// TIA Portal project "Project4" (V15.1)

(* hardware
DEVICE "S7-1200 station_2"  S7-1200 Station
   slot 0: "Rack_0"  S7-1200 Rack  Rack  V1.0
   slot 1: "CLP2_TESTING"  CPU 1214C DC/DC/DC  6ES7 214-1AG40-0XB0  V4.2
      slot 3: "AQ 1x12BIT_1"  AQ1 signal board  6ES7 232-4HA30-0XB0  V1.0
   slot 2: "DI 8/DQ 8x24VDC_1"  SM 1223 DI8/DQ8 x 24VDC  6ES7 223-1BH30-0XB0  V1.0
*)

// ===== PLC "CLP2_TESTING"  CPU 1214C DC/DC/DC =====

VAR_GLOBAL   // PLC tag table "Default tag table"
   "PART_AV" AT %I0.0 : Bool;
   "B2" AT %I0.1 : Bool;
   "B4" AT %I0.2 : Bool;
   "B5" AT %I0.3 : Bool;
   "1B1" AT %I0.4 : Bool;
   "1B2" AT %I0.5 : Bool;
   "2B1" AT %I0.6 : Bool;
   "IP_FI" AT %I0.7 : Bool;
   "Bot_Start" AT %I8.0 : Bool;
   "Bot_Stop" AT %I8.1 : Bool;
   "Bot_Reset" AT %I8.3 : Bool;
   "Desce_Elevador" AT %Q0.0 : Bool;
   "Sobe_Elevador" AT %Q0.1 : Bool;
   "Empurra_Peça" AT %Q0.2 : Bool;
   "Rampa" AT %Q0.3 : Bool;
   "IP_N_FO" AT %Q0.7 : Bool;
   "LED_Start" AT %Q8.0 : Bool;
   "LED_Reset" AT %Q8.1 : Bool;
   "LED_Q1" AT %Q8.2 : Bool;
   "LED_Q2" AT %Q8.3 : Bool;
   "void" AT %M57.0 : Bool;
   "Chega_Peça" AT %M0.0 : Bool;
   "Subida_Liberada" AT %M0.1 : Bool;
   "void2" AT %M57.1 : Bool;
   "Elevador_Em_Cima" AT %M0.3 : Bool;
   "void3" AT %M57.2 : Bool;
   "Elevador_Embaixo" AT %M0.4 : Bool;
   "void4" AT %M57.3 : Bool;
   "Pistão_Recuou" AT %M0.5 : Bool;
   "void5" AT %M57.4 : Bool;
   "Altura_Certa" AT %M0.6 : Bool;
   "Prox.Bancada_Liberou" AT %M0.7 : Bool;
   "void6" AT %M57.5 : Bool;
   "void7" AT %M57.6 : Bool;
   "void8" AT %M57.7 : Bool;
   "Start" AT %M1.0 : Bool;
   "Reset" AT %M1.1 : Bool;
   "Stop" AT %M1.2 : Bool;
   "Elevador_Subindo" AT %M2.0 : Bool;
   "Testando_Altura" AT %M2.1 : Bool;
   "Elevador_Descendo_c_Peça" AT %M2.2 : Bool;
   "Empurrando_Peça" AT %M2.3 : Bool;
   "Elevador_Descendo_Vazio" AT %M2.4 : Bool;
   "Descartando_Peça" AT %M2.5 : Bool;
   "Elevador_Livre" AT %M2.6 : Bool;
   "Contador_Descarte" AT %MW4 : Int;
   "Rampa_Desl" AT %M3.0 : Bool;
   "Rampa_Lig" AT %M3.1 : Bool;
   "Prox_Bancada_Livre" AT %M3.2 : Bool;
   "Parado" AT %M3.3 : Bool;
   "Resetando_Elevador" AT %M3.4 : Bool;
   "Pronto" AT %M3.5 : Bool;
   "Tem_Peça" AT %M2.7 : Bool;
   "T1" AT %M4.0 : Bool;
   "T2" AT %M4.1 : Bool;
   "T3" AT %M4.2 : Bool;
   "T4" AT %M4.3 : Bool;
   "T5" AT %M4.4 : Bool;
   "T6" AT %M4.5 : Bool;
   "T7" AT %M4.6 : Bool;
   "T8" AT %M6.0 : Bool;
   "T9" AT %M6.1 : Bool;
   "T10" AT %M6.2 : Bool;
   "T11" AT %M6.3 : Bool;
   "T12" AT %M6.4 : Bool;
   "T13" AT %M6.5 : Bool;
   "T14" AT %M6.6 : Bool;
   "T15" AT %M6.7 : Bool;
   "T16" AT %M7.0 : Bool;
   "T17" AT %M7.1 : Bool;
   "T18" AT %M7.2 : Bool;
   "T19" AT %M7.3 : Bool;
   "T20" AT %M7.4 : Bool;
   "T21" AT %M7.5 : Bool;
   "T22" AT %M7.6 : Bool;
   "T23" AT %M7.7 : Bool;
   "T24" AT %M8.0 : Bool;
   "T0" AT %M8.1 : Bool;
   "Fim_Reset" AT %M8.2 : Bool;
   "T25" AT %M8.3 : Bool;
   "Memo_Inicialização" AT %M58.0 : Bool;
   "T26" AT %M8.4 : Bool;
   "Resetando_Pistão" AT %M3.6 : Bool;
   "T27" AT %M8.5 : Bool;
   "Tag_1" AT %M58.1 : Bool;
   "Pistão_Recuado" AT %M58.2 : Bool;
END_VAR

// folder: System blocks/Program resources

DATA_BLOCK "IEC_Timer_0_DB_2"   // DB1
{ S7_Optimized_Access := 'TRUE' }
AUTHOR : Simatic
FAMILY : IEC
NAME : IEC_TMR
VERSION : 1.0
// stored: InstanceOfName IEC_TIMER
"IEC_TIMER"
BEGIN
END_DATA_BLOCK

DATA_BLOCK "IEC_Timer_0_DB"   // DB2
{ S7_Optimized_Access := 'TRUE' }
AUTHOR : Simatic
FAMILY : IEC
NAME : IEC_TMR
VERSION : 1.0
// stored: InstanceOfName IEC_TIMER
"IEC_TIMER"
BEGIN
END_DATA_BLOCK

DATA_BLOCK "IEC_Counter_0_DB_1"   // DB3
{ S7_Optimized_Access := 'TRUE' }
AUTHOR : Simatic
FAMILY : IEC
NAME : CNTR
VERSION : 1.0
// stored: InstanceOfName IEC_COUNTER
"IEC_COUNTER"
BEGIN
END_DATA_BLOCK

DATA_BLOCK "IEC_Timer_0_DB_1"   // DB4
{ S7_Optimized_Access := 'TRUE' }
AUTHOR : Simatic
FAMILY : IEC
NAME : IEC_TMR
VERSION : 1.0
// stored: InstanceOfName IEC_TIMER
"IEC_TIMER"
BEGIN
END_DATA_BLOCK

// folder: (top level)

FUNCTION "Eventos Externos" : Void   // FC1, LAD
{ S7_Optimized_Access := 'TRUE' }
VERSION : 0.1
   VAR_TEMP   // added for the SCL form of the ladder/FBD networks
      _w1 : Bool;
      _w2 : Bool;
      _w3 : Bool;
      _w4 : Bool;
      _w5 : Bool;
      _w6 : Bool;
   END_VAR
BEGIN

REGION Network 1
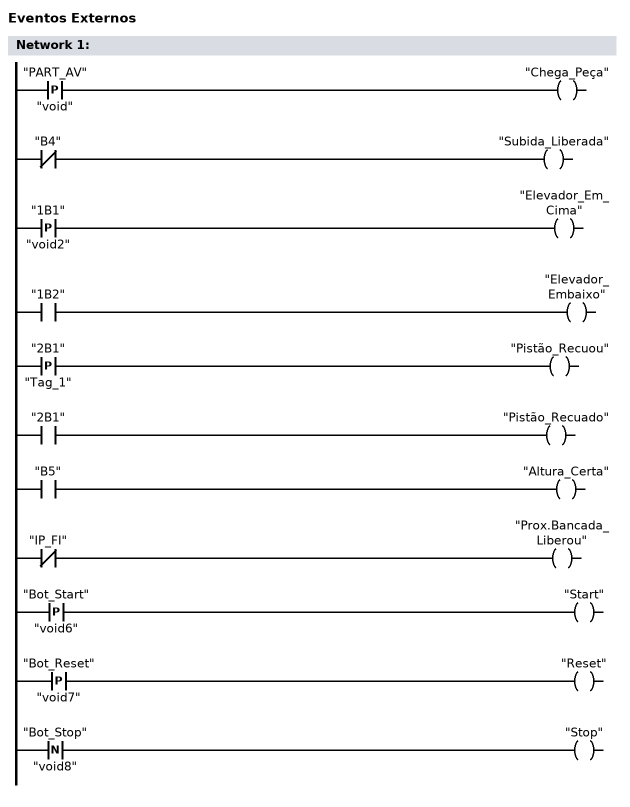
   RUNG wire#powerrail
      P_Contact(operand := "PART_AV", bit := "void")
      Coil( "Chega_Peça" )
   END_RUNG
   RUNG wire#powerrail
      I_Contact( "B4" )
      Coil( "Subida_Liberada" )
   END_RUNG
   RUNG wire#powerrail
      P_Contact(operand := "1B1", bit := "void2")
      Coil( "Elevador_Em_Cima" )
   END_RUNG
   RUNG wire#powerrail
      Contact( "1B2" )
      Coil( "Elevador_Embaixo" )
   END_RUNG
   RUNG wire#powerrail
      P_Contact(operand := "2B1", bit := "Tag_1")
      Coil( "Pistão_Recuou" )
   END_RUNG
   RUNG wire#powerrail
      Contact( "2B1" )
      Coil( "Pistão_Recuado" )
   END_RUNG
   RUNG wire#powerrail
      Contact( "B5" )
      Coil( "Altura_Certa" )
   END_RUNG
   RUNG wire#powerrail
      I_Contact( "IP_FI" )
      Coil( "Prox.Bancada_Liberou" )
   END_RUNG
   RUNG wire#powerrail
      P_Contact(operand := "Bot_Start", bit := "void6")
      Coil( "Start" )
   END_RUNG
   RUNG wire#powerrail
      P_Contact(operand := "Bot_Reset", bit := "void7")
      Coil( "Reset" )
   END_RUNG
   RUNG wire#powerrail
      N_Contact(operand := "Bot_Stop", bit := "void8")
      Coil( "Stop" )
   END_RUNG
   // the same network as SCL:
   #_w1 := "PART_AV" AND NOT "void";   // rising edge of "PART_AV"
   "void" := "PART_AV";
   "Chega_Peça" := #_w1;
   "Subida_Liberada" := NOT "B4";
   #_w2 := "1B1" AND NOT "void2";   // rising edge of "1B1"
   "void2" := "1B1";
   "Elevador_Em_Cima" := #_w2;
   "Elevador_Embaixo" := "1B2";
   #_w3 := "2B1" AND NOT "Tag_1";   // rising edge of "2B1"
   "Tag_1" := "2B1";
   "Pistão_Recuou" := #_w3;
   "Pistão_Recuado" := "2B1";
   "Altura_Certa" := "B5";
   "Prox.Bancada_Liberou" := NOT "IP_FI";
   #_w4 := "Bot_Start" AND NOT "void6";   // rising edge of "Bot_Start"
   "void6" := "Bot_Start";
   "Start" := #_w4;
   #_w5 := "Bot_Reset" AND NOT "void7";   // rising edge of "Bot_Reset"
   "void7" := "Bot_Reset";
   "Reset" := #_w5;
   #_w6 := NOT "Bot_Stop" AND "void8";   // falling edge of "Bot_Stop"
   "void8" := "Bot_Stop";
   "Stop" := #_w6;
END_REGION
END_FUNCTION

FUNCTION "Condicoes_Disparo" : Void   // FC2, LAD
{ S7_Optimized_Access := 'TRUE' }
VERSION : 0.1
BEGIN

REGION Network 1
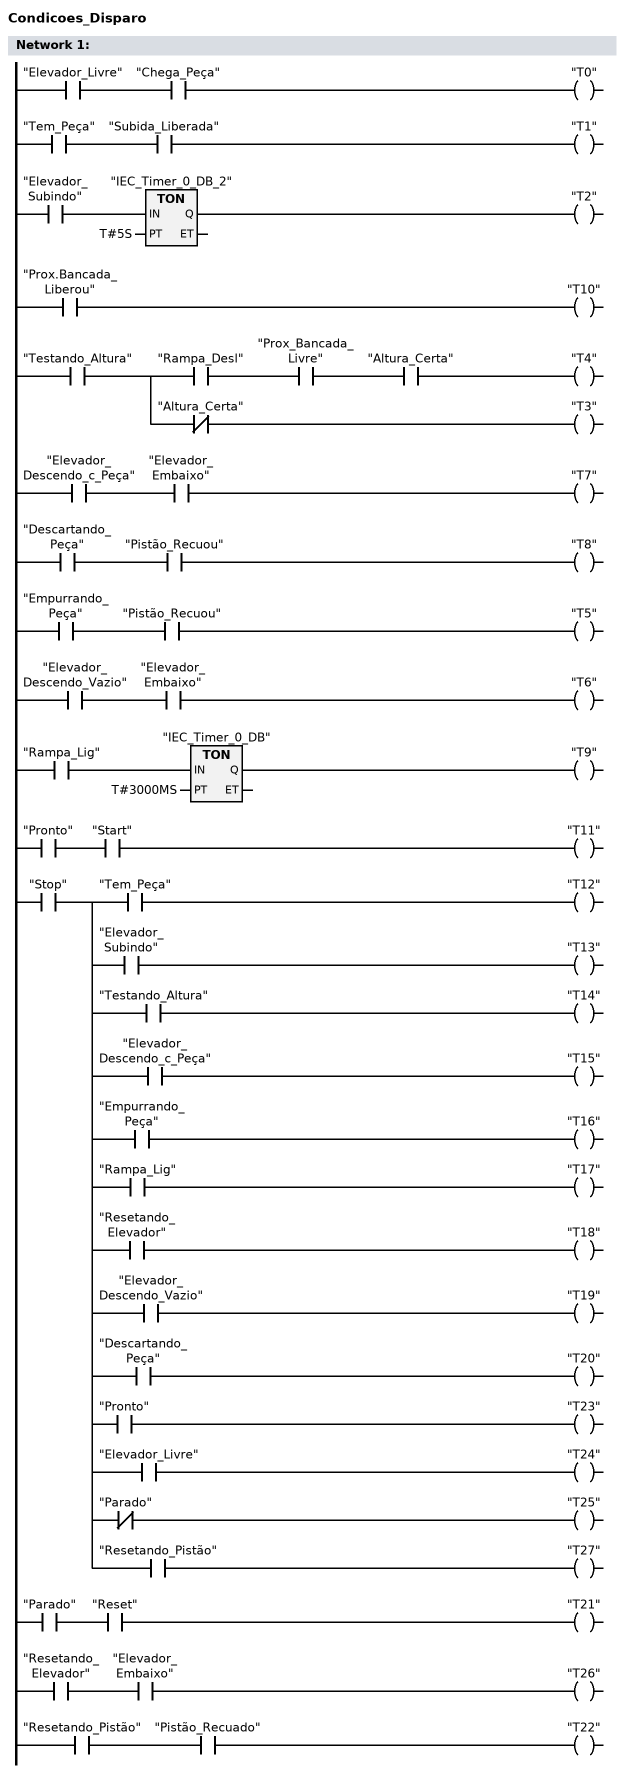
   "T0" := "Elevador_Livre" AND "Chega_Peça";
   "T1" := "Tem_Peça" AND "Subida_Liberada";
   "IEC_Timer_0_DB_2".TON(IN := "Elevador_Subindo", PT := T#5S);
   "T2" := "IEC_Timer_0_DB_2".Q;
   "T10" := "Prox.Bancada_Liberou";
   "T4" := "Testando_Altura" AND "Rampa_Desl" AND "Prox_Bancada_Livre" AND "Altura_Certa";
   "T3" := "Testando_Altura" AND NOT "Altura_Certa";
   "T7" := "Elevador_Descendo_c_Peça" AND "Elevador_Embaixo";
   "T8" := "Descartando_Peça" AND "Pistão_Recuou";
   "T5" := "Empurrando_Peça" AND "Pistão_Recuou";
   "T6" := "Elevador_Descendo_Vazio" AND "Elevador_Embaixo";
   "IEC_Timer_0_DB".TON(IN := "Rampa_Lig", PT := T#3000MS);
   "T9" := "IEC_Timer_0_DB".Q;
   "T11" := "Pronto" AND "Start";
   "T12" := "Stop" AND "Tem_Peça";
   "T13" := "Stop" AND "Elevador_Subindo";
   "T14" := "Stop" AND "Testando_Altura";
   "T15" := "Stop" AND "Elevador_Descendo_c_Peça";
   "T16" := "Stop" AND "Empurrando_Peça";
   "T17" := "Stop" AND "Rampa_Lig";
   "T18" := "Stop" AND "Resetando_Elevador";
   "T19" := "Stop" AND "Elevador_Descendo_Vazio";
   "T20" := "Stop" AND "Descartando_Peça";
   "T23" := "Stop" AND "Pronto";
   "T24" := "Stop" AND "Elevador_Livre";
   "T25" := "Stop" AND NOT "Parado";
   "T27" := "Stop" AND "Resetando_Pistão";
   "T21" := "Parado" AND "Reset";
   "T26" := "Resetando_Elevador" AND "Elevador_Embaixo";
   "T22" := "Resetando_Pistão" AND "Pistão_Recuado";
END_REGION
END_FUNCTION

FUNCTION "Dinamica Fichas" : Void   // FC3, LAD
{ S7_Optimized_Access := 'TRUE' }
VERSION : 0.1
BEGIN

REGION Network 1
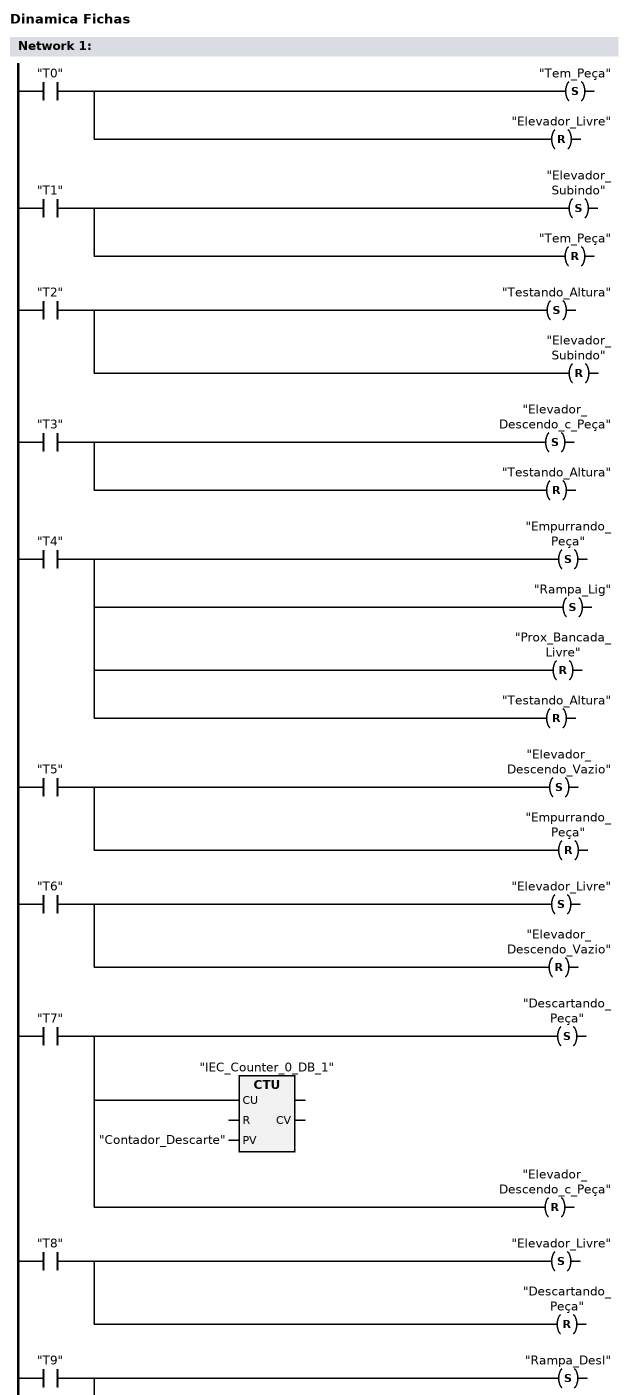
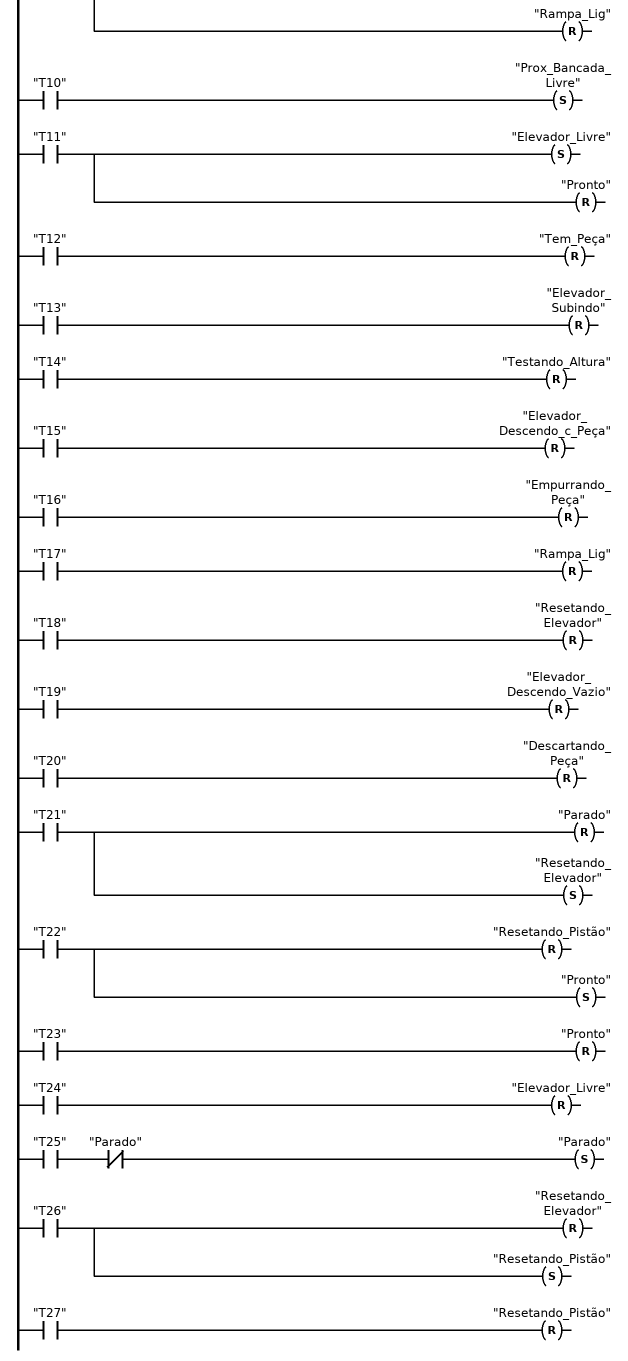
   IF "T0" THEN
       "Tem_Peça" := TRUE;
       "Elevador_Livre" := FALSE;
   END_IF;
   IF "T1" THEN
       "Elevador_Subindo" := TRUE;
       "Tem_Peça" := FALSE;
   END_IF;
   IF "T2" THEN
       "Testando_Altura" := TRUE;
       "Elevador_Subindo" := FALSE;
   END_IF;
   IF "T3" THEN
       "Elevador_Descendo_c_Peça" := TRUE;
       "Testando_Altura" := FALSE;
   END_IF;
   IF "T4" THEN
       "Empurrando_Peça" := TRUE;
       "Rampa_Lig" := TRUE;
       "Prox_Bancada_Livre" := FALSE;
       "Testando_Altura" := FALSE;
   END_IF;
   IF "T5" THEN
       "Elevador_Descendo_Vazio" := TRUE;
       "Empurrando_Peça" := FALSE;
   END_IF;
   IF "T6" THEN
       "Elevador_Livre" := TRUE;
       "Elevador_Descendo_Vazio" := FALSE;
   END_IF;
   IF "T7" THEN "Descartando_Peça" := TRUE; END_IF;
   "IEC_Counter_0_DB_1".CTU(CU := "T7", PV := "Contador_Descarte");
   IF "T7" THEN "Elevador_Descendo_c_Peça" := FALSE; END_IF;
   IF "T8" THEN
       "Elevador_Livre" := TRUE;
       "Descartando_Peça" := FALSE;
   END_IF;
   IF "T9" THEN
       "Rampa_Desl" := TRUE;
       "Rampa_Lig" := FALSE;
   END_IF;
   IF "T10" THEN "Prox_Bancada_Livre" := TRUE; END_IF;
   IF "T11" THEN
       "Elevador_Livre" := TRUE;
       "Pronto" := FALSE;
   END_IF;
   IF "T12" THEN "Tem_Peça" := FALSE; END_IF;
   IF "T13" THEN "Elevador_Subindo" := FALSE; END_IF;
   IF "T14" THEN "Testando_Altura" := FALSE; END_IF;
   IF "T15" THEN "Elevador_Descendo_c_Peça" := FALSE; END_IF;
   IF "T16" THEN "Empurrando_Peça" := FALSE; END_IF;
   IF "T17" THEN "Rampa_Lig" := FALSE; END_IF;
   IF "T18" THEN "Resetando_Elevador" := FALSE; END_IF;
   IF "T19" THEN "Elevador_Descendo_Vazio" := FALSE; END_IF;
   IF "T20" THEN "Descartando_Peça" := FALSE; END_IF;
   IF "T21" THEN
       "Parado" := FALSE;
       "Resetando_Elevador" := TRUE;
   END_IF;
   IF "T22" THEN
       "Resetando_Pistão" := FALSE;
       "Pronto" := TRUE;
   END_IF;
   IF "T23" THEN "Pronto" := FALSE; END_IF;
   IF "T24" THEN "Elevador_Livre" := FALSE; END_IF;
   IF "T25" AND NOT "Parado" THEN "Parado" := TRUE; END_IF;
   IF "T26" THEN
       "Resetando_Elevador" := FALSE;
       "Resetando_Pistão" := TRUE;
   END_IF;
   IF "T27" THEN "Resetando_Pistão" := FALSE; END_IF;
END_REGION
END_FUNCTION

FUNCTION "Inicialização" : Void   // FC4, LAD
{ S7_Optimized_Access := 'TRUE' }
VERSION : 0.1
   VAR_TEMP   // added for the SCL form of the ladder/FBD networks
      _w1 : Bool;
   END_VAR
BEGIN

REGION Network 1
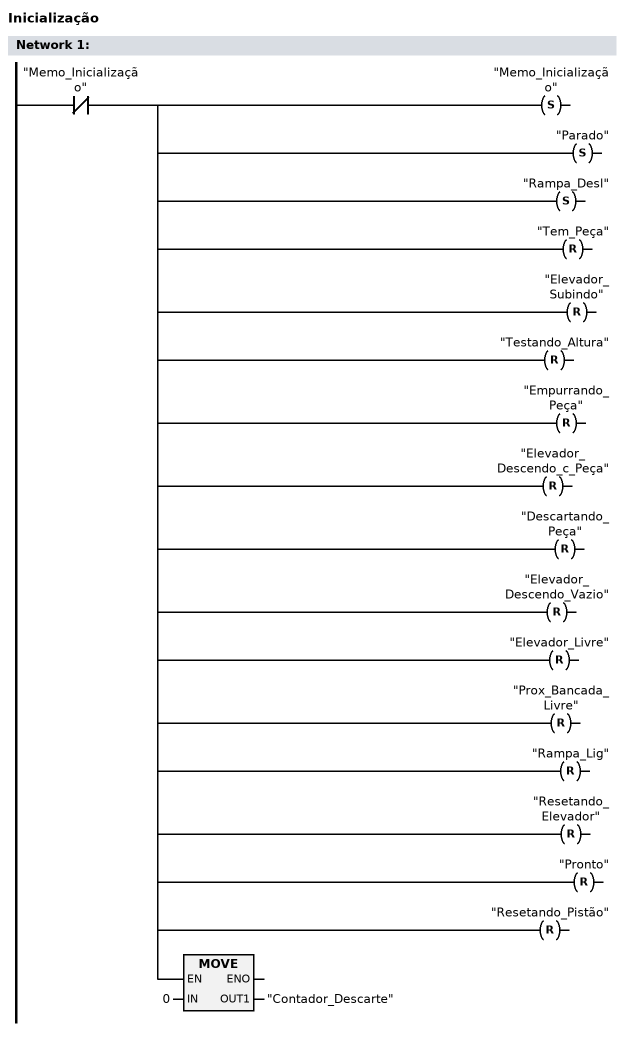
   RUNG wire#powerrail
      I_Contact( "Memo_Inicialização" )
      wire#w1
      S_Coil( "Memo_Inicialização" )
   END_RUNG
   RUNG wire#w1
      S_Coil( "Parado" )
   END_RUNG
   RUNG wire#w1
      S_Coil( "Rampa_Desl" )
   END_RUNG
   RUNG wire#w1
      R_Coil( "Tem_Peça" )
   END_RUNG
   RUNG wire#w1
      R_Coil( "Elevador_Subindo" )
   END_RUNG
   RUNG wire#w1
      R_Coil( "Testando_Altura" )
   END_RUNG
   RUNG wire#w1
      R_Coil( "Empurrando_Peça" )
   END_RUNG
   RUNG wire#w1
      R_Coil( "Elevador_Descendo_c_Peça" )
   END_RUNG
   RUNG wire#w1
      R_Coil( "Descartando_Peça" )
   END_RUNG
   RUNG wire#w1
      R_Coil( "Elevador_Descendo_Vazio" )
   END_RUNG
   RUNG wire#w1
      R_Coil( "Elevador_Livre" )
   END_RUNG
   RUNG wire#w1
      R_Coil( "Prox_Bancada_Livre" )
   END_RUNG
   RUNG wire#w1
      R_Coil( "Rampa_Lig" )
   END_RUNG
   RUNG wire#w1
      R_Coil( "Resetando_Elevador" )
   END_RUNG
   RUNG wire#w1
      R_Coil( "Pronto" )
   END_RUNG
   RUNG wire#w1
      R_Coil( "Resetando_Pistão" )
   END_RUNG
   RUNG wire#w1
      Move(in := 0, out1 => "Contador_Descarte")
   END_RUNG
   // the same network as SCL:
   #_w1 := NOT "Memo_Inicialização";
   IF #_w1 THEN
       "Memo_Inicialização" := TRUE;
       "Parado" := TRUE;
       "Rampa_Desl" := TRUE;
       "Tem_Peça" := FALSE;
       "Elevador_Subindo" := FALSE;
       "Testando_Altura" := FALSE;
       "Empurrando_Peça" := FALSE;
       "Elevador_Descendo_c_Peça" := FALSE;
       "Descartando_Peça" := FALSE;
       "Elevador_Descendo_Vazio" := FALSE;
       "Elevador_Livre" := FALSE;
       "Prox_Bancada_Livre" := FALSE;
       "Rampa_Lig" := FALSE;
       "Resetando_Elevador" := FALSE;
       "Pronto" := FALSE;
       "Resetando_Pistão" := FALSE;
       "Contador_Descarte" := 0;
   END_IF;
END_REGION
END_FUNCTION

FUNCTION "Ações" : Void   // FC5, LAD
{ S7_Optimized_Access := 'TRUE' }
VERSION : 0.1
BEGIN

REGION Network 1
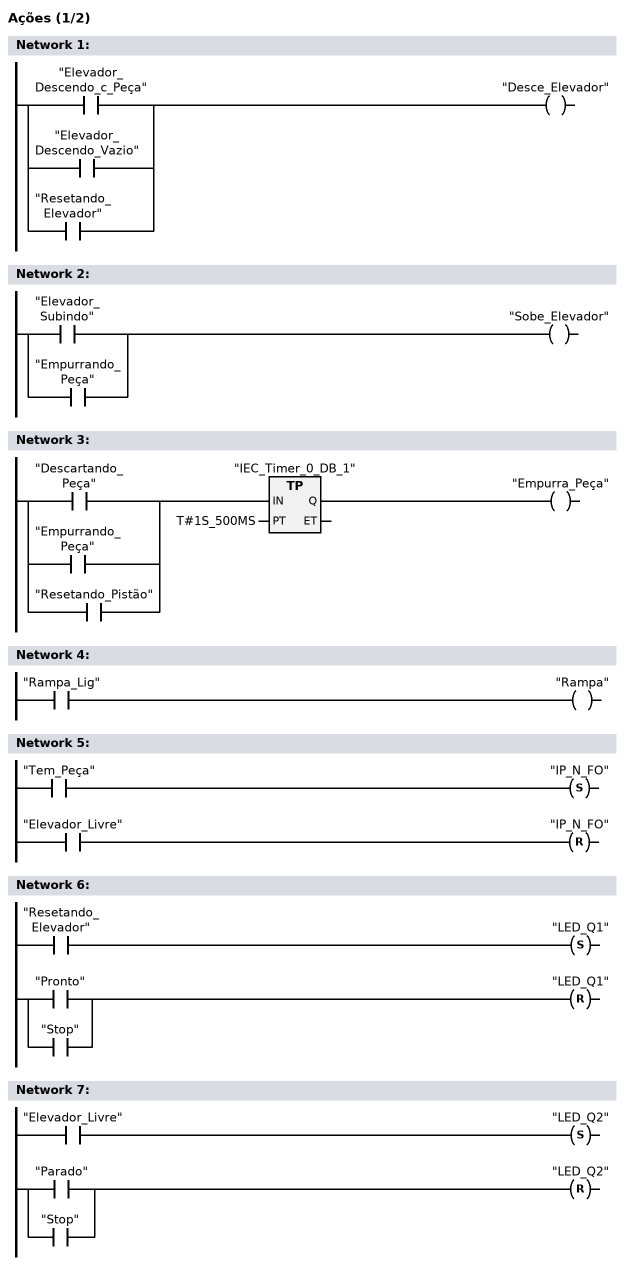
   RUNG wire#powerrail
      Contact( "Elevador_Descendo_c_Peça" )
      wire#w1
      Coil( "Desce_Elevador" )
   END_RUNG
   RUNG wire#powerrail
      Contact( "Elevador_Descendo_Vazio" )
   END_RUNG wire#w1
   RUNG wire#powerrail
      Contact( "Resetando_Elevador" )
   END_RUNG wire#w1
   // the same network as SCL:
   "Desce_Elevador" := "Elevador_Descendo_c_Peça" OR "Elevador_Descendo_Vazio" OR "Resetando_Elevador";
END_REGION

REGION Network 2
   RUNG wire#powerrail
      Contact( "Elevador_Subindo" )
      wire#w1
      Coil( "Sobe_Elevador" )
   END_RUNG
   RUNG wire#powerrail
      Contact( "Empurrando_Peça" )
   END_RUNG wire#w1
   // the same network as SCL:
   "Sobe_Elevador" := "Elevador_Subindo" OR "Empurrando_Peça";
END_REGION

REGION Network 3
   "IEC_Timer_0_DB_1".TP(IN := "Descartando_Peça" OR "Empurrando_Peça" OR "Resetando_Pistão", PT := T#1S_500MS);
   "Empurra_Peça" := "IEC_Timer_0_DB_1".Q;
END_REGION

REGION Network 4
   RUNG wire#powerrail
      Contact( "Rampa_Lig" )
      Coil( "Rampa" )
   END_RUNG
   // the same network as SCL:
   "Rampa" := "Rampa_Lig";
END_REGION

REGION Network 5
   RUNG wire#powerrail
      Contact( "Tem_Peça" )
      S_Coil( "IP_N_FO" )
   END_RUNG
   RUNG wire#powerrail
      Contact( "Elevador_Livre" )
      R_Coil( "IP_N_FO" )
   END_RUNG
   // the same network as SCL:
   IF "Tem_Peça" THEN "IP_N_FO" := TRUE; END_IF;
   IF "Elevador_Livre" THEN "IP_N_FO" := FALSE; END_IF;
END_REGION

REGION Network 6
   RUNG wire#powerrail
      Contact( "Resetando_Elevador" )
      S_Coil( "LED_Q1" )
   END_RUNG
   RUNG wire#powerrail
      Contact( "Pronto" )
      wire#w1
      R_Coil( "LED_Q1" )
   END_RUNG
   RUNG wire#powerrail
      Contact( "Stop" )
   END_RUNG wire#w1
   // the same network as SCL:
   IF "Resetando_Elevador" THEN "LED_Q1" := TRUE; END_IF;
   IF "Pronto" OR "Stop" THEN "LED_Q1" := FALSE; END_IF;
END_REGION

REGION Network 7
   RUNG wire#powerrail
      Contact( "Elevador_Livre" )
      S_Coil( "LED_Q2" )
   END_RUNG
   RUNG wire#powerrail
      Contact( "Parado" )
      wire#w1
      R_Coil( "LED_Q2" )
   END_RUNG
   RUNG wire#powerrail
      Contact( "Stop" )
   END_RUNG wire#w1
   // the same network as SCL:
   IF "Elevador_Livre" THEN "LED_Q2" := TRUE; END_IF;
   IF "Parado" OR "Stop" THEN "LED_Q2" := FALSE; END_IF;
END_REGION

REGION Network 8
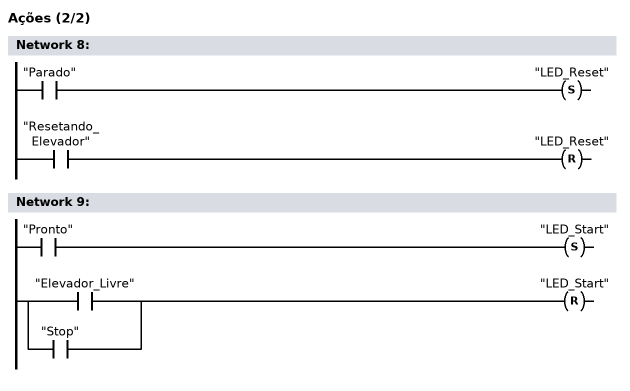
   RUNG wire#powerrail
      Contact( "Parado" )
      S_Coil( "LED_Reset" )
   END_RUNG
   RUNG wire#powerrail
      Contact( "Resetando_Elevador" )
      R_Coil( "LED_Reset" )
   END_RUNG
   // the same network as SCL:
   IF "Parado" THEN "LED_Reset" := TRUE; END_IF;
   IF "Resetando_Elevador" THEN "LED_Reset" := FALSE; END_IF;
END_REGION

REGION Network 9
   RUNG wire#powerrail
      Contact( "Pronto" )
      S_Coil( "LED_Start" )
   END_RUNG
   RUNG wire#powerrail
      Contact( "Elevador_Livre" )
      wire#w1
      R_Coil( "LED_Start" )
   END_RUNG
   RUNG wire#powerrail
      Contact( "Stop" )
   END_RUNG wire#w1
   // the same network as SCL:
   IF "Pronto" THEN "LED_Start" := TRUE; END_IF;
   IF "Elevador_Livre" OR "Stop" THEN "LED_Start" := FALSE; END_IF;
END_REGION
END_FUNCTION

ORGANIZATION_BLOCK "Main"   // OB1, LAD, ProgramCycle
TITLE = "Main Program Sweep (Cycle)"
{ S7_Optimized_Access := 'TRUE' }
VERSION : 0.1
   VAR_INPUT
      Initial_Call : Bool;   // Initial call of this OB
      Remanence : Bool;   // =True, if remanent data are available
   END_VAR
BEGIN

REGION Network 1
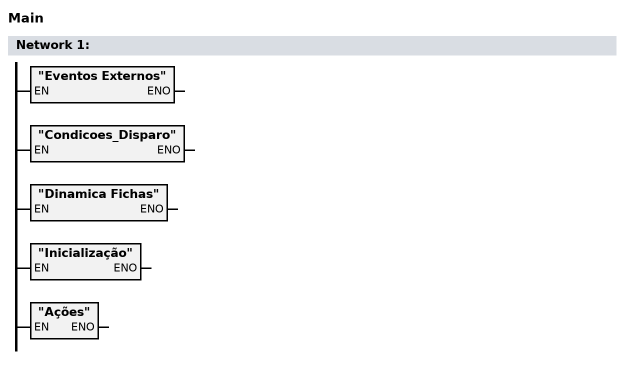
   RUNG wire#powerrail
      "Eventos Externos"()
   END_RUNG
   RUNG wire#powerrail
      "Condicoes_Disparo"()
   END_RUNG
   RUNG wire#powerrail
      "Dinamica Fichas"()
   END_RUNG
   RUNG wire#powerrail
      "Inicialização"()
   END_RUNG
   RUNG wire#powerrail
      "Ações"()
   END_RUNG
   // the same network as SCL:
   "Eventos Externos"();
   "Condicoes_Disparo"();
   "Dinamica Fichas"();
   "Inicialização"();
   "Ações"();
END_REGION
END_ORGANIZATION_BLOCK